NodeFactory.AddNodeAsPrototype('Vision/Basic Container Operations/F_VN_InsertIntoContainer/F_VN_InsertIntoContainer_DINT', node_F_VN_InsertIntoContainer_DINT);
NodeFactory.AddNodeAsPrototype('Vision/Basic Container Operations/F_VN_InsertIntoContainer/F_VN_InsertIntoContainer_INT', node_F_VN_InsertIntoContainer_INT);
NodeFactory.AddNodeAsPrototype('Vision/Basic Container Operations/F_VN_InsertIntoContainer/F_VN_InsertIntoContainer_ITcVnContainer', node_F_VN_InsertIntoContainer_ITcVnContainer);
//NodeFactory.AddNodeAsPrototype('Vision/Basic Container Operations/F_VN_InsertIntoContainer/F_VN_InsertIntoContainer_ITcVnForwardIterator', node_F_VN_InsertIntoContainer_ITcVnForwardIterator);
NodeFactory.AddNodeAsPrototype('Vision/Basic Container Operations/F_VN_InsertIntoContainer/F_VN_InsertIntoContainer_ITcVnImage', node_F_VN_InsertIntoContainer_ITcVnImage);
NodeFactory.AddNodeAsPrototype('Vision/Basic Container Operations/F_VN_InsertIntoContainer/F_VN_InsertIntoContainer_LREAL', node_F_VN_InsertIntoContainer_LREAL);
NodeFactory.AddNodeAsPrototype('Vision/Basic Container Operations/F_VN_InsertIntoContainer/F_VN_InsertIntoContainer_REAL', node_F_VN_InsertIntoContainer_REAL);
NodeFactory.AddNodeAsPrototype('Vision/Basic Container Operations/F_VN_InsertIntoContainer/F_VN_InsertIntoContainer_SINT', node_F_VN_InsertIntoContainer_SINT);
NodeFactory.AddNodeAsPrototype('Vision/Basic Container Operations/F_VN_InsertIntoContainer/F_VN_InsertIntoContainer_TcVnDMatch', node_F_VN_InsertIntoContainer_TcVnDMatch);
NodeFactory.AddNodeAsPrototype('Vision/Basic Container Operations/F_VN_InsertIntoContainer/F_VN_InsertIntoContainer_TcVnKeyPoint', node_F_VN_InsertIntoContainer_TcVnKeyPoint);
NodeFactory.AddNodeAsPrototype('Vision/Basic Container Operations/F_VN_InsertIntoContainer/F_VN_InsertIntoContainer_TcVnPoint2_DINT', node_F_VN_InsertIntoContainer_TcVnPoint2_DINT);
NodeFactory.AddNodeAsPrototype('Vision/Basic Container Operations/F_VN_InsertIntoContainer/F_VN_InsertIntoContainer_TcVnPoint2_LREAL', node_F_VN_InsertIntoContainer_TcVnPoint2_LREAL);
NodeFactory.AddNodeAsPrototype('Vision/Basic Container Operations/F_VN_InsertIntoContainer/F_VN_InsertIntoContainer_TcVnPoint2_REAL', node_F_VN_InsertIntoContainer_TcVnPoint2_REAL);
NodeFactory.AddNodeAsPrototype('Vision/Basic Container Operations/F_VN_InsertIntoContainer/F_VN_InsertIntoContainer_TcVnPoint3_LREAL', node_F_VN_InsertIntoContainer_TcVnPoint3_LREAL);
NodeFactory.AddNodeAsPrototype('Vision/Basic Container Operations/F_VN_InsertIntoContainer/F_VN_InsertIntoContainer_TcVnPoint3_REAL', node_F_VN_InsertIntoContainer_TcVnPoint3_REAL);
NodeFactory.AddNodeAsPrototype('Vision/Basic Container Operations/F_VN_InsertIntoContainer/F_VN_InsertIntoContainer_TcVnRectangle_DINT', node_F_VN_InsertIntoContainer_TcVnRectangle_DINT);
NodeFactory.AddNodeAsPrototype('Vision/Basic Container Operations/F_VN_InsertIntoContainer/F_VN_InsertIntoContainer_TcVnVector2_DINT', node_F_VN_InsertIntoContainer_TcVnVector2_DINT);
NodeFactory.AddNodeAsPrototype('Vision/Basic Container Operations/F_VN_InsertIntoContainer/F_VN_InsertIntoContainer_TcVnVector2_INT', node_F_VN_InsertIntoContainer_TcVnVector2_INT);
NodeFactory.AddNodeAsPrototype('Vision/Basic Container Operations/F_VN_InsertIntoContainer/F_VN_InsertIntoContainer_TcVnVector2_REAL', node_F_VN_InsertIntoContainer_TcVnVector2_REAL);
NodeFactory.AddNodeAsPrototype('Vision/Basic Container Operations/F_VN_InsertIntoContainer/F_VN_InsertIntoContainer_TcVnVector2_SINT', node_F_VN_InsertIntoContainer_TcVnVector2_SINT);
NodeFactory.AddNodeAsPrototype('Vision/Basic Container Operations/F_VN_InsertIntoContainer/F_VN_InsertIntoContainer_TcVnVector2_UINT', node_F_VN_InsertIntoContainer_TcVnVector2_UINT);
NodeFactory.AddNodeAsPrototype('Vision/Basic Container Operations/F_VN_InsertIntoContainer/F_VN_InsertIntoContainer_TcVnVector2_USINT', node_F_VN_InsertIntoContainer_TcVnVector2_USINT);
NodeFactory.AddNodeAsPrototype('Vision/Basic Container Operations/F_VN_InsertIntoContainer/F_VN_InsertIntoContainer_TcVnVector3_INT', node_F_VN_InsertIntoContainer_TcVnVector3_INT);
NodeFactory.AddNodeAsPrototype('Vision/Basic Container Operations/F_VN_InsertIntoContainer/F_VN_InsertIntoContainer_TcVnVector3_REAL', node_F_VN_InsertIntoContainer_TcVnVector3_REAL);
NodeFactory.AddNodeAsPrototype('Vision/Basic Container Operations/F_VN_InsertIntoContainer/F_VN_InsertIntoContainer_TcVnVector3_SINT', node_F_VN_InsertIntoContainer_TcVnVector3_SINT);
NodeFactory.AddNodeAsPrototype('Vision/Basic Container Operations/F_VN_InsertIntoContainer/F_VN_InsertIntoContainer_TcVnVector3_UINT', node_F_VN_InsertIntoContainer_TcVnVector3_UINT);
NodeFactory.AddNodeAsPrototype('Vision/Basic Container Operations/F_VN_InsertIntoContainer/F_VN_InsertIntoContainer_TcVnVector3_USINT', node_F_VN_InsertIntoContainer_TcVnVector3_USINT);
NodeFactory.AddNodeAsPrototype('Vision/Basic Container Operations/F_VN_InsertIntoContainer/F_VN_InsertIntoContainer_TcVnVector4_DINT', node_F_VN_InsertIntoContainer_TcVnVector4_DINT);
NodeFactory.AddNodeAsPrototype('Vision/Basic Container Operations/F_VN_InsertIntoContainer/F_VN_InsertIntoContainer_TcVnVector4_INT', node_F_VN_InsertIntoContainer_TcVnVector4_INT);
NodeFactory.AddNodeAsPrototype('Vision/Basic Container Operations/F_VN_InsertIntoContainer/F_VN_InsertIntoContainer_TcVnVector4_LREAL', node_F_VN_InsertIntoContainer_TcVnVector4_LREAL);
NodeFactory.AddNodeAsPrototype('Vision/Basic Container Operations/F_VN_InsertIntoContainer/F_VN_InsertIntoContainer_TcVnVector4_SINT', node_F_VN_InsertIntoContainer_TcVnVector4_SINT);
NodeFactory.AddNodeAsPrototype('Vision/Basic Container Operations/F_VN_InsertIntoContainer/F_VN_InsertIntoContainer_TcVnVector4_UINT', node_F_VN_InsertIntoContainer_TcVnVector4_UINT);
NodeFactory.AddNodeAsPrototype('Vision/Basic Container Operations/F_VN_InsertIntoContainer/F_VN_InsertIntoContainer_TcVnVector4_USINT', node_F_VN_InsertIntoContainer_TcVnVector4_USINT);
NodeFactory.AddNodeAsPrototype('Vision/Basic Container Operations/F_VN_InsertIntoContainer/F_VN_InsertIntoContainer_UDINT', node_F_VN_InsertIntoContainer_UDINT);
NodeFactory.AddNodeAsPrototype('Vision/Basic Container Operations/F_VN_InsertIntoContainer/F_VN_InsertIntoContainer_UINT', node_F_VN_InsertIntoContainer_UINT);
NodeFactory.AddNodeAsPrototype('Vision/Basic Container Operations/F_VN_InsertIntoContainer/F_VN_InsertIntoContainer_ULINT', node_F_VN_InsertIntoContainer_ULINT);
NodeFactory.AddNodeAsPrototype('Vision/Basic Container Operations/F_VN_InsertIntoContainer/F_VN_InsertIntoContainer_USINT', node_F_VN_InsertIntoContainer_USINT);

NodeFactory.AddNodeAsPrototype('Vision/Basic Container Operations/F_VN_SetAt/F_VN_SetAt_DINT', node_F_VN_SetAt_DINT);
NodeFactory.AddNodeAsPrototype('Vision/Basic Container Operations/F_VN_SetAt/F_VN_SetAt_INT', node_F_VN_SetAt_INT);
NodeFactory.AddNodeAsPrototype('Vision/Basic Container Operations/F_VN_SetAt/F_VN_SetAt_ITcVnContainer', node_F_VN_SetAt_ITcVnContainer);
NodeFactory.AddNodeAsPrototype('Vision/Basic Container Operations/F_VN_SetAt/F_VN_SetAt_ITcVnImage', node_F_VN_SetAt_ITcVnImage);
NodeFactory.AddNodeAsPrototype('Vision/Basic Container Operations/F_VN_SetAt/F_VN_SetAt_LREAL', node_F_VN_SetAt_LREAL);
NodeFactory.AddNodeAsPrototype('Vision/Basic Container Operations/F_VN_SetAt/F_VN_SetAt_REAL', node_F_VN_SetAt_REAL);
NodeFactory.AddNodeAsPrototype('Vision/Basic Container Operations/F_VN_SetAt/F_VN_SetAt_SINT', node_F_VN_SetAt_SINT);
NodeFactory.AddNodeAsPrototype('Vision/Basic Container Operations/F_VN_SetAt/F_VN_SetAt_TcVnDMatch', node_F_VN_SetAt_TcVnDMatch);
NodeFactory.AddNodeAsPrototype('Vision/Basic Container Operations/F_VN_SetAt/F_VN_SetAt_TcVnKeyPoint', node_F_VN_SetAt_TcVnKeyPoint);
NodeFactory.AddNodeAsPrototype('Vision/Basic Container Operations/F_VN_SetAt/F_VN_SetAt_TcVnPoint2_DINT', node_F_VN_SetAt_TcVnPoint2_DINT);
NodeFactory.AddNodeAsPrototype('Vision/Basic Container Operations/F_VN_SetAt/F_VN_SetAt_TcVnPoint2_LREAL', node_F_VN_SetAt_TcVnPoint2_LREAL);
NodeFactory.AddNodeAsPrototype('Vision/Basic Container Operations/F_VN_SetAt/F_VN_SetAt_TcVnPoint2_REAL', node_F_VN_SetAt_TcVnPoint2_REAL);
NodeFactory.AddNodeAsPrototype('Vision/Basic Container Operations/F_VN_SetAt/F_VN_SetAt_TcVnPoint3_LREAL', node_F_VN_SetAt_TcVnPoint3_LREAL);
NodeFactory.AddNodeAsPrototype('Vision/Basic Container Operations/F_VN_SetAt/F_VN_SetAt_TcVnPoint3_REAL', node_F_VN_SetAt_TcVnPoint3_REAL);
NodeFactory.AddNodeAsPrototype('Vision/Basic Container Operations/F_VN_SetAt/F_VN_SetAt_TcVnRectangle_DINT', node_F_VN_SetAt_TcVnRectangle_DINT);
NodeFactory.AddNodeAsPrototype('Vision/Basic Container Operations/F_VN_SetAt/F_VN_SetAt_TcVnVector2_DINT', node_F_VN_SetAt_TcVnVector2_DINT);
NodeFactory.AddNodeAsPrototype('Vision/Basic Container Operations/F_VN_SetAt/F_VN_SetAt_TcVnVector2_INT', node_F_VN_SetAt_TcVnVector2_INT);
NodeFactory.AddNodeAsPrototype('Vision/Basic Container Operations/F_VN_SetAt/F_VN_SetAt_TcVnVector2_REAL', node_F_VN_SetAt_TcVnVector2_REAL);
NodeFactory.AddNodeAsPrototype('Vision/Basic Container Operations/F_VN_SetAt/F_VN_SetAt_TcVnVector2_SINT', node_F_VN_SetAt_TcVnVector2_SINT);
NodeFactory.AddNodeAsPrototype('Vision/Basic Container Operations/F_VN_SetAt/F_VN_SetAt_TcVnVector2_UINT', node_F_VN_SetAt_TcVnVector2_UINT);
NodeFactory.AddNodeAsPrototype('Vision/Basic Container Operations/F_VN_SetAt/F_VN_SetAt_TcVnVector2_USINT', node_F_VN_SetAt_TcVnVector2_USINT);
NodeFactory.AddNodeAsPrototype('Vision/Basic Container Operations/F_VN_SetAt/F_VN_SetAt_TcVnVector3_INT', node_F_VN_SetAt_TcVnVector3_INT);
NodeFactory.AddNodeAsPrototype('Vision/Basic Container Operations/F_VN_SetAt/F_VN_SetAt_TcVnVector3_REAL', node_F_VN_SetAt_TcVnVector3_REAL);
NodeFactory.AddNodeAsPrototype('Vision/Basic Container Operations/F_VN_SetAt/F_VN_SetAt_TcVnVector3_SINT', node_F_VN_SetAt_TcVnVector3_SINT);
NodeFactory.AddNodeAsPrototype('Vision/Basic Container Operations/F_VN_SetAt/F_VN_SetAt_TcVnVector3_UINT', node_F_VN_SetAt_TcVnVector3_UINT);
NodeFactory.AddNodeAsPrototype('Vision/Basic Container Operations/F_VN_SetAt/F_VN_SetAt_TcVnVector3_USINT', node_F_VN_SetAt_TcVnVector3_USINT);
NodeFactory.AddNodeAsPrototype('Vision/Basic Container Operations/F_VN_SetAt/F_VN_SetAt_TcVnVector4_DINT', node_F_VN_SetAt_TcVnVector4_DINT);
NodeFactory.AddNodeAsPrototype('Vision/Basic Container Operations/F_VN_SetAt/F_VN_SetAt_TcVnVector4_INT', node_F_VN_SetAt_TcVnVector4_INT);
NodeFactory.AddNodeAsPrototype('Vision/Basic Container Operations/F_VN_SetAt/F_VN_SetAt_TcVnVector4_LREAL', node_F_VN_SetAt_TcVnVector4_LREAL);
NodeFactory.AddNodeAsPrototype('Vision/Basic Container Operations/F_VN_SetAt/F_VN_SetAt_TcVnVector4_SINT', node_F_VN_SetAt_TcVnVector4_SINT);
NodeFactory.AddNodeAsPrototype('Vision/Basic Container Operations/F_VN_SetAt/F_VN_SetAt_TcVnVector4_UINT', node_F_VN_SetAt_TcVnVector4_UINT);
NodeFactory.AddNodeAsPrototype('Vision/Basic Container Operations/F_VN_SetAt/F_VN_SetAt_TcVnVector4_USINT', node_F_VN_SetAt_TcVnVector4_USINT);
NodeFactory.AddNodeAsPrototype('Vision/Basic Container Operations/F_VN_SetAt/F_VN_SetAt_UDINT', node_F_VN_SetAt_UDINT);
NodeFactory.AddNodeAsPrototype('Vision/Basic Container Operations/F_VN_SetAt/F_VN_SetAt_UINT', node_F_VN_SetAt_UINT);
NodeFactory.AddNodeAsPrototype('Vision/Basic Container Operations/F_VN_SetAt/F_VN_SetAt_ULINT', node_F_VN_SetAt_ULINT);
NodeFactory.AddNodeAsPrototype('Vision/Basic Container Operations/F_VN_SetAt/F_VN_SetAt_USINT', node_F_VN_SetAt_USINT);

NodeFactory.AddNodeAsPrototype('Vision/Basic Container Operations/F_VN_GetNumberOfElements', node_F_VN_GetNumberOfElements);

// Basic Image Operations
NodeFactory.AddNodeAsPrototype('Vision/Basic Image Operations/F_VN_CopyImage', node_F_VN_CopyImage);
NodeFactory.AddNodeAsPrototype('Vision/Basic Image Operations/F_VN_GetImageChannel', node_F_VN_GetImageChannel);
NodeFactory.AddNodeAsPrototype('Vision/Basic Image Operations/F_VN_GetImageHeight', node_F_VN_GetImageHeight);
NodeFactory.AddNodeAsPrototype('Vision/Basic Image Operations/F_VN_GetImageInfo', node_F_VN_GetImageInfo);
NodeFactory.AddNodeAsPrototype('Vision/Basic Image Operations/F_VN_GetImageWidth', node_F_VN_GetImageWidth);
NodeFactory.AddNodeAsPrototype('Vision/Basic Image Operations/F_VN_GetPixelFormat', node_F_VN_GetPixelFormat);
NodeFactory.AddNodeAsPrototype('Vision/Basic Image Operations/F_VN_SetRoi', node_F_VN_SetRoi);
//NodeFactory.AddNodeAsPrototype('Vision/Basic Image Operations/F_VN_SetRoi_TcVnRectangle_DINT', node_F_VN_SetRoi_TcVnRectangle_DINT);
 
// Code Quality

// Code Reading

// Constants
NodeFactory.AddNodeAsPrototype('Vision/Constants/RGBA_BLACK', node_RGBA_BLACK);
NodeFactory.AddNodeAsPrototype('Vision/Constants/RGBA_RED', node_RGBA_RED);
NodeFactory.AddNodeAsPrototype('Vision/Constants/RGBA_YELLOW', node_RGBA_YELLOW);
NodeFactory.AddNodeAsPrototype('Vision/Constants/RGBA_GREEN', node_RGBA_GREEN);
NodeFactory.AddNodeAsPrototype('Vision/Constants/RGBA_CYAN', node_RGBA_CYAN);
NodeFactory.AddNodeAsPrototype('Vision/Constants/RGBA_BLUE', node_RGBA_BLUE);
NodeFactory.AddNodeAsPrototype('Vision/Constants/RGBA_MAGENTA', node_RGBA_MAGENTA);
NodeFactory.AddNodeAsPrototype('Vision/Constants/RGBA_WHITE', node_RGBA_WHITE);

// Container Statistics

// Contour Analysis
NodeFactory.AddNodeAsPrototype('Vision/Contour Analysis/F_VN_FitLine', node_F_VN_FitLine);

// Control Functions
    
// Drawing
NodeFactory.AddNodeAsPrototype('Vision/Drawing/F_VN_DrawContours', node_F_VN_DrawContours);
NodeFactory.AddNodeAsPrototype('Vision/Drawing/F_VN_DrawLine', node_F_VN_DrawLine);
NodeFactory.AddNodeAsPrototype('Vision/Drawing/F_VN_DrawLine_TcVnVector4_LREAL', node_F_VN_DrawLine_TcVnVector4_LREAL);
NodeFactory.AddNodeAsPrototype('Vision/Drawing/F_VN_PutLabel', node_F_VN_PutLabel);
NodeFactory.AddNodeAsPrototype('Vision/Drawing/F_VN_PutText', node_F_VN_PutText);

// Fourier Analysis

// Geometric and Coordinate Transformations
NodeFactory.AddNodeAsPrototype('Vision/Geometric and Coordinate Transformations/F_VN_FlipImage', node_F_VN_FlipImage);

// Image Analysis
NodeFactory.AddNodeAsPrototype('Vision/Image Analysis/Object Detection/F_VN_DetectBlobs', node_F_VN_DetectBlobs);

// Image Color and Contrast Processing
NodeFactory.AddNodeAsPrototype('Vision/Image Color and Contrast Processing/F_VN_ApplyColorMap', node_F_VN_ApplyColorMap);
NodeFactory.AddNodeAsPrototype('Vision/Image Color and Contrast Processing/F_VN_ConvertColorSpace', node_F_VN_ConvertColorSpace);
NodeFactory.AddNodeAsPrototype('Vision/Image Color and Contrast Processing/F_VN_GenerateColorMap', node_F_VN_GenerateColorMap);

// Image Filtering
NodeFactory.AddNodeAsPrototype('Vision/Image Filtering/F_VN_BoxFilter', node_F_VN_BoxFilter);
NodeFactory.AddNodeAsPrototype('Vision/Image Filtering/F_VN_GaussianFilter', node_F_VN_GaussianFilter);
NodeFactory.AddNodeAsPrototype('Vision/Image Filtering/F_VN_LaplacianFilter', node_F_VN_LaplacianFilter);
    
// Image Segmentation
NodeFactory.AddNodeAsPrototype('Vision/Image Segmentation/F_VN_Threshold', node_F_VN_Threshold);

// Keypoint Features

// Machine Learning

// Measurement
NodeFactory.AddNodeAsPrototype('Vision/Measurement/F_VN_LocateEdge', node_F_VN_LocateEdge);

// Miscellaneous

// OCR

// Texture Analysis
END_METHOD

END_FUNCTION_BLOCK

// VisionPack
{attribute 'linkalways'} 
{attribute 'no_explicit_call' := 'This FB is a CLASS and must be accessed using methods or properties'}
{attribute 'enable_dynamic_creation'}
FUNCTION_BLOCK VisionPack IMPLEMENTS I_GraphPack
VAR
	visionDatatypePack : VisionDatatypePack;
	visionNodePack : VisionNodePack;
END_VAR

METHOD RegisterWithDatatypes
VAR_INPUT
	Datatypes : I_Datatypes;
END_VAR
visionDatatypePack.RegisterWithDatatypes(Datatypes);
END_METHOD

METHOD PUBLIC RegisterWithNodeFactory
VAR_INPUT
	NodeFactory : I_NodeFactory;
END_VAR
visionNodePack.RegisterWithNodeFactory(NodeFactory);
END_METHOD

END_FUNCTION_BLOCK
